{attribute 'to_string'}
{attribute 'qualified_only'}
{attribute 'strict'}
TYPE nHP_Axis_BrakeMode:
(
	BrakeMode_Automatic := 0,
    BrakeMode_Lock:= 1,
    BrakeMode_Unlock:= 2
);
END_TYPE

(* stored: Version 1.1.0.1, ProductVersion 3.1.4024.12
   EnumerationTextList nHP_Axis_BrakeMode: Id {5bcfef8f-a323-4cf5-b072-ce93735ba1fd} *)
